(* CODESYS project GarageDoor_student.project2.project

Project tree, tasks and I/O mapping:
  Device : CODESYS Control Win V3, 3S - Smart Software Solutions GmbH, version 3.5.16.20
    application Application
      libraries: Standard, * (System); Util, * (System)
      task MainTask (cyclic, interval t#10ms, priority 1) calls Model, PLC_PRG
      visualisation Visualization
      image pool ImagePool
      program Model [ST]
      program PLC_PRG [FBD]
  text list GlobalTextList
  5ce3da45-db07-42e7-a21c-a00fff4ed8f6|E:\inside_garage_lowlow.png
  5ce3da45-db07-42e7-a21c-a00fff4ed8f6|E:\garage_lowlow.png
  5ce3da45-db07-42e7-a21c-a00fff4ed8f6|E:\door_lowlow.png
*)

// Device/Application/Model
PROGRAM Model
VAR CONSTANT
	cycleTime :DWORD :=10;
	integSpeed :REAL :=0.5;
	maxSpeed :REAL :=2.0;
END_VAR
VAR
	// Inputs
	motor :BOOL :=FALSE;
	direction :BOOL :=FALSE;
	// Outputs
	button :BOOL :=FALSE;
	downSensor :BOOL;
	upSensor :BOOL;
	// States
	STOP :BOOL :=TRUE;
	UP :BOOL :=FALSE;
	DOWN :BOOL :=FALSE;
	// Other variables
	posDoor :REAL :=0.0;
	speedDoor :REAL :=0.0;
	doIntegral :INTEGRAL;
	inBetween :BOOL :=FALSE;
	doorMoving :BOOL :=FALSE;
END_VAR

// Read inputs
motor := PLC_PRG.motor;
direction := PLC_PRG.direction;

// State 1: Stop
IF (UP AND (upSensor OR NOT(motor))) OR (DOWN AND (downSensor OR NOT(motor))) THEN
	STOP := TRUE;
	UP := FALSE;
	DOWN := FALSE;
END_IF

// State 2: Going up
IF (motor AND NOT(direction) AND NOT(upSensor)) THEN
	UP := TRUE;
	STOP := FALSE;
	DOWN := FALSE;
END_IF

// State 3: Going down
IF motor AND direction AND NOT(downSensor) THEN
	DOWN := TRUE;
	STOP := FALSE;
	UP := FALSE;
END_IF

// Perform actions from states
IF STOP THEN
	doIntegral(RESET:=STOP);
	doorMoving := FALSE;
END_IF
IF UP THEN
	doIntegral(IN:=-integSpeed,TM:=cycleTime,RESET:=STOP,OUT=>speedDoor);
	doorMoving := TRUE;
END_IF
IF DOWN THEN
	doIntegral(IN:=integSpeed,TM:=cycleTime,RESET:=STOP,OUT=>speedDoor);
	doorMoving := TRUE;
END_IF

// Check actions of states
// Set upper limit for garage door
IF posDoor + speedDoor < -285.0 THEN
	posDoor := -285.0;
	speedDoor := 0.0;
	upSensor := TRUE;
	inBetween := FALSE;
END_IF
// Set lower limit for garage door
IF posDoor + speedDoor > 0.0 THEN
	posDoor := 0.0;
	speedDoor := 0.0;
	downSensor := TRUE;
	inBetween := FALSE;
END_IF
// Move the door if not in STOP state, also limit integral output
IF NOT(STOP) THEN
		IF speedDoor >= maxSpeed THEN
			posDoor := posDoor + maxSpeed;
		ELSIF speedDoor <= -maxSpeed THEN
			posDoor := posDoor -maxSpeed;
		ELSE
			posDoor := posDoor + speedDoor;
		END_IF
END_IF
// Turn yellow light when door stops in between upper and lower sensor
IF posDoor > -285.0 AND posDOOR < 0.0 THEN
	inBetween := TRUE;
	upSensor := FALSE;
	downSensor := FALSE;
END_IF
	

// Write to outputs
PLC_PRG.button := button;
PLC_PRG.sensor_lower := downSensor;
PLC_PRG.sensor_upper := upSensor;

END_PROGRAM

// Device/Application/PLC_PRG
PROGRAM PLC_PRG
VAR_INPUT
	// input
	button:BOOL;
	sensor_lower:BOOL;
	sensor_upper:BOOL;
END_VAR
VAR_OUTPUT
	// output
	motor:BOOL := true;
	direction:BOOL := true;
END_VAR
VAR
	click: R_TRIG;
	switch: R_TRIG;
	A: R_TRIG;
	B: R_TRIG;
	C: R_TRIG;
END_VAR
VAR // added by the converter: edge detectors and wires of the graphical bodies
    _rt1, _rt2, _rt3, _rt4 : R_TRIG;
END_VAR

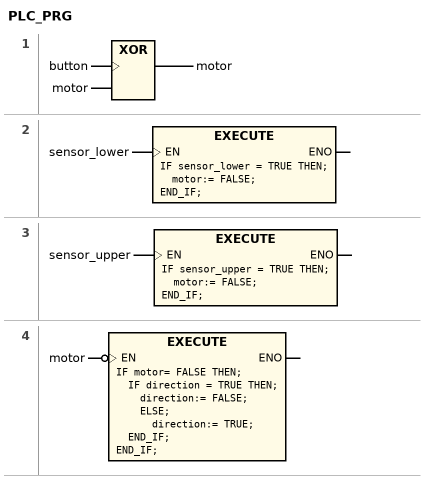
// NETWORK 1
_rt1(CLK := button);
motor := _rt1.Q XOR motor;

// NETWORK 2
_rt2(CLK := sensor_lower);
IF _rt2.Q THEN
    IF sensor_lower = TRUE THEN;
    	motor:= FALSE;
    END_IF;
END_IF

// NETWORK 3
_rt3(CLK := sensor_upper);
IF _rt3.Q THEN
    IF sensor_upper = TRUE THEN;
    	motor:= FALSE;
    END_IF;
END_IF

// NETWORK 4
_rt4(CLK := NOT motor);
IF _rt4.Q THEN
    IF motor= FALSE THEN;
    	IF direction = TRUE THEN;
    		direction:= FALSE;
    		ELSE;
    			direction:= TRUE;
    	END_IF;
    END_IF;
END_IF

END_PROGRAM

// Device/Application/Visualization
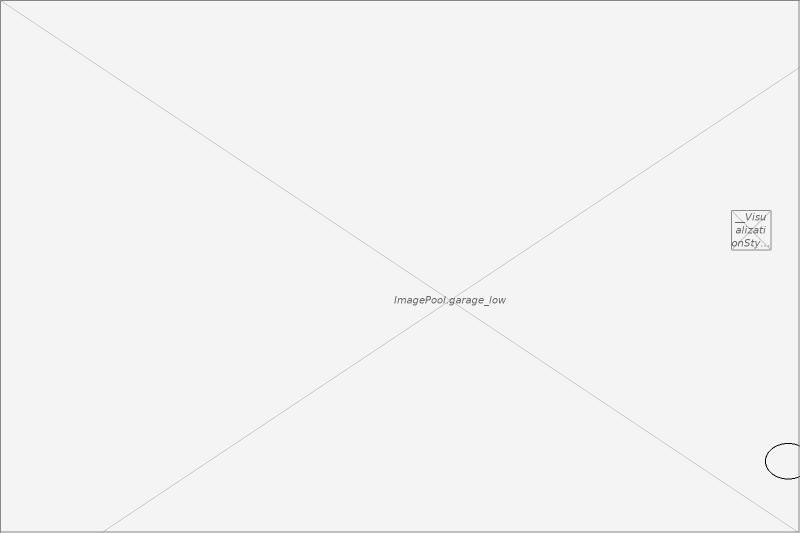
VISUALIZATION Visualization  // 800x533
    Image (149,188 578x338), image: ImagePool.inside_garage_low
    Image (151,213 569x285), image: ImagePool.door_low
        p2738717112: Model.posDoor
    Image (0,0 900x600), image: ImagePool.garage_low
    Image (731,210 40x40)
    Ellipse (765,443 46x36)
        tap Model.button
    Image (731,210 40x40), invisible if: NOT(Model.downSensor OR Model.upSensor)
    Image (731,210 40x40), invisible if: NOT(Model.doorMoving)
    Image (731,210 40x40), invisible if: NOT(Model.inBetween AND Model.STOP)
END_VISUALIZATION
